// TIA Portal V18 export
FUNCTION_BLOCK "RollerV3"   // FB2, LAD
TITLE = Description:
{ S7_Optimized_Access := 'TRUE' }
VERSION : 0.1
// How to operate and control the roller:
// Roller is controled by inputs in WebDB: Mode, SetSpeed, Direction, OffsetSpeed. To start the roller use Start_Roller and to stop use Stop_Roller.
// 
// Mode descriptions:
// 0 - Controlling the roller by just turning it ON/OFF
// 1 - Basic speed control of the roller with 0-100%
// 2 - Direct speed control based on Y axis velocity. Not useful for printing, but might help in the development process to observe roller system inertia.
// 3 - Setting relative surface velocity (powder to roller). There is no control loop. Could be used for testing the feature before evaluating.
// 
// E-STOP - always check!
// stored: AutoNumber true, IsIECCheckEnabled false, IsRetainMemResEnabled false, MemoryReserve 100, SetENOAutomatically false, UDAEnableTagReadback false
   VAR_INPUT
      "E-STOP" : Bool;
      SystemON : Bool;
      Mode : Int;   // 0 - ON/OFF; 1 - Set Max Speed; 2 - Automatic Yvel=Rvel; 3 - Automatic vel dif
      SetSpeed : Real;   // %
      DirectionLeftRight : Bool;
      Offsetspeed : DInt;
      YAxisVelocity : DInt;
      Roller_HW_address : HW_HSC;
      DoorSensors : Bool;
   END_VAR
   VAR_OUTPUT
      WebDBRollerOutput : Bool;
      RollerDirection : Bool;   // 1 - Clockwise; 0 - Counterclockwise
      RollerLinearVelocity : DInt;   // Microns Per Sec
      RollerRPM : Real;
      RollerRPM_Measured : Real;
   END_VAR
   VAR_IN_OUT
      WebDBStart : Bool;
      WebDBStop : Bool;
   END_VAR
   VAR
      RollerSetReset : Bool;
      RollerFullPower : Bool;
      RollerHalfPower : Bool;
      RollerActive : Bool;
      RollerSpeedInputGeneral { ExternalAccessible := 'False'; ExternalVisible := 'False'; ExternalWritable := 'False'} : Real;   // %
      RollerSpeedInputPID : Real;
      RollerManualValue : Int;
      Direction_Plus { ExternalAccessible := 'False'; ExternalVisible := 'False'; ExternalWritable := 'False'} : Bool;   // Clockwise
      Direction_Minus { ExternalAccessible := 'False'; ExternalVisible := 'False'; ExternalWritable := 'False'} : Bool;   // Counterclockwise
      PulseSignalMeasurement : DWord;
      MaintenanceM3DirDis : Bool := true;
      MaintenanceSkipPID : Bool := true;
      MaintenanceAutomaticDifVel : Bool;   // Change automatic mode from Yvel=Rvel to Difference
      MaintenanceRollerON : Bool;
      RollerDirectionInt_last : Int;
      Roller_RPM_Send_last : Real;
      RollerSetReset_M : Bool;
      RollerSetReset_M2 : Bool;
      hscData : HSC_Period;
   END_VAR
   VAR_TEMP
      DirectionMinusInternal : Bool;
      OffsetSpeedInternal : DInt;
      YAxisVelocityInternal : DInt;
      Roller_Speed_ConvRPM : Real;
      Roller_Speed_ConvPercInput : Real;
      Roller_Speed_ConvDEGSEC : Real;
      Roller_PWM_NormOutput : Real;
      Roller_ConvLinearPerDeg : DInt;
      Roller_Conv_M1_Norm : Real;
      Roller_Conv_M1_Scale : Real;
      Roller_Conv_M2_YvelocityconvRPS : Real;
      Roller_Conv_M2_YvelocityconvRPM : Real;
      Roller_Conv_M3_LinVel : DInt;
      Roller_Conv_M3_Rps : Real;
      Roller_Conv_M3_Rpm : Real;
      Roller_Send_Conv : Real;
      Roller_RPM_Send : Real;
      Roller_RPM_SendRev : Real;
      Roller_Circumference : DInt;   // [microns]
      Roller_Direction_Internal : Bool;
      RollerMinRPMRev : Real;
      RollerDirectionInt : Int;
      ex_vel : Bool;
      RollerDEGPS_send : Real;
      RPMchanged : Bool;
      DirectionChanged : Bool;
      haltAxis : Bool;
   END_VAR
   VAR CONSTANT
      RollerMotorMaxSpeed : Real := 200.0;   // RPM
      MotorToRollerGearRatio : Real := 1.0;   // Belt transmission ratio
      RPMtoDEGSEC : Real := 6.0;   // RPM to Degress per Second conversion factor
      RollerDiameter : DInt := 50000;   // Diameter in microns
      LinearRollerSpeedFactor : Real;   // To convert rotation to linear speed
      RollerPWMPeriod : Int := 10000;
      RollerMinRPM : Real := 5.0;
   END_VAR
   // hscData.EnHSC := TRUE;
   // hscData.EnPeriod := false;
   // hscData.NewPeriod := 1000;
   VAR_TEMP   // added for the SCL form of the ladder/FBD networks
      _w1 : Bool;
      _w2 : Bool;
   END_VAR
BEGIN

REGION Network 1: Roller ON and Speed Control
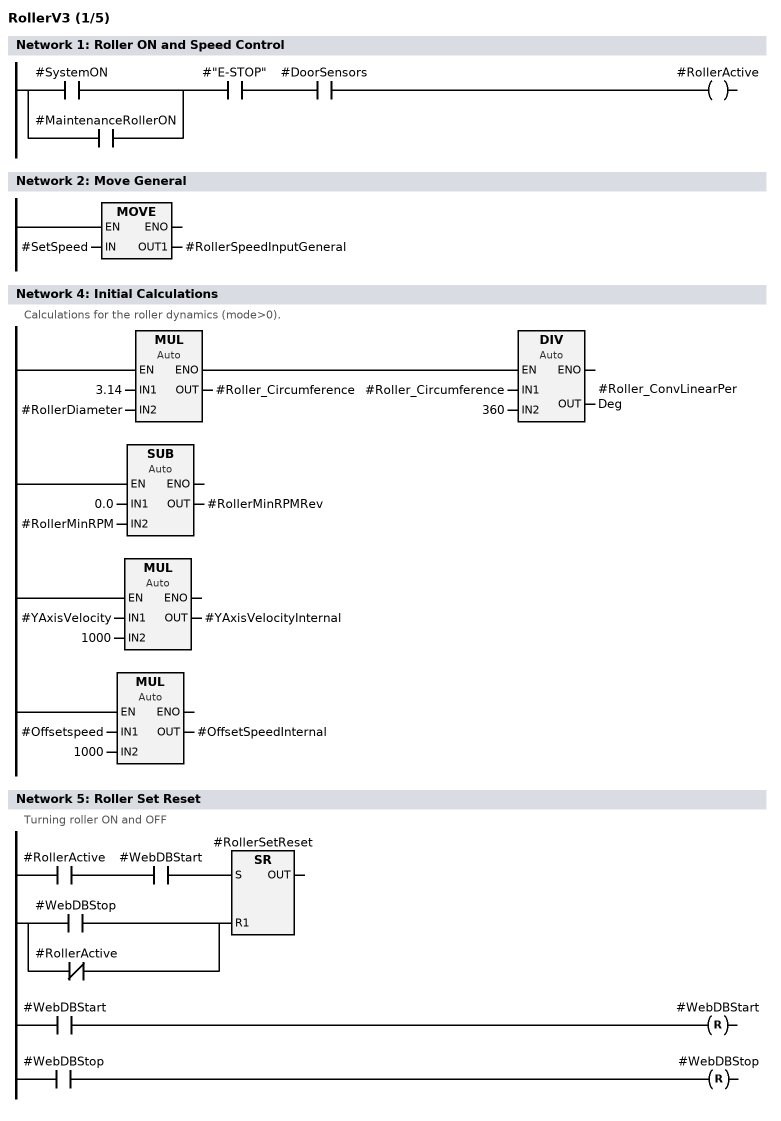
   RUNG wire#powerrail
      Contact( #SystemON )
      wire#w1
      Contact( #"E-STOP" )
      Contact( #DoorSensors )
      Coil( #RollerActive )
   END_RUNG
   RUNG wire#powerrail
      Contact( #MaintenanceRollerON )
   END_RUNG wire#w1
   // the same network as SCL:
   #RollerActive := (#SystemON OR #MaintenanceRollerON) AND #"E-STOP" AND #DoorSensors;
END_REGION

REGION Network 2: Move General
   RUNG wire#powerrail
      Move(in := #SetSpeed, out1 => #RollerSpeedInputGeneral)
   END_RUNG
   // the same network as SCL:
   #RollerSpeedInputGeneral := #SetSpeed;
END_REGION

REGION Network 3: Roller Direction
END_REGION

REGION Network 4: Initial Calculations
   // Calculations for the roller dynamics (mode>0).
   RUNG wire#powerrail
      Mul(in1 := 3.14, in2 := #RollerDiameter, out => #Roller_Circumference)
      Div(in1 := #Roller_Circumference, in2 := 360, out => #Roller_ConvLinearPerDeg)
   END_RUNG
   RUNG wire#powerrail
      Sub(in1 := 0.0, in2 := #RollerMinRPM, out => #RollerMinRPMRev)
   END_RUNG
   RUNG wire#powerrail
      Mul(in1 := #YAxisVelocity, in2 := 1000, out => #YAxisVelocityInternal)
   END_RUNG
   RUNG wire#powerrail
      Mul(in1 := #Offsetspeed, in2 := 1000, out => #OffsetSpeedInternal)
   END_RUNG
   // the same network as SCL:
   #Roller_Circumference := 3.14 * #RollerDiameter;
   #Roller_ConvLinearPerDeg := #Roller_Circumference / 360;
   #RollerMinRPMRev := 0.0 - #RollerMinRPM;
   #YAxisVelocityInternal := #YAxisVelocity * 1000;
   #OffsetSpeedInternal := #Offsetspeed * 1000;
END_REGION

REGION Network 5: Roller Set Reset
   // Turning roller ON and OFF
   RUNG wire#powerrail
      Contact( #RollerActive )
      Contact( #WebDBStart )
      S_SR(operand := #RollerSetReset, r1 := wire#w1)
   END_RUNG
   RUNG wire#powerrail
      Contact( #WebDBStop )
   END_RUNG wire#w1
   RUNG wire#powerrail
      I_Contact( #RollerActive )
   END_RUNG wire#w1
   RUNG wire#powerrail
      Contact( #WebDBStart )
      R_Coil( #WebDBStart )
   END_RUNG
   RUNG wire#powerrail
      Contact( #WebDBStop )
      R_Coil( #WebDBStop )
   END_RUNG
   // the same network as SCL:
   IF #RollerActive AND #WebDBStart THEN
       #RollerSetReset := TRUE;   // SR flip-flop
   END_IF;
   IF #WebDBStop OR NOT #RollerActive THEN #RollerSetReset := FALSE; END_IF;
   IF #WebDBStart THEN #WebDBStart := FALSE; END_IF;
   IF #WebDBStop THEN #WebDBStop := FALSE; END_IF;
END_REGION

REGION Network 6: PID
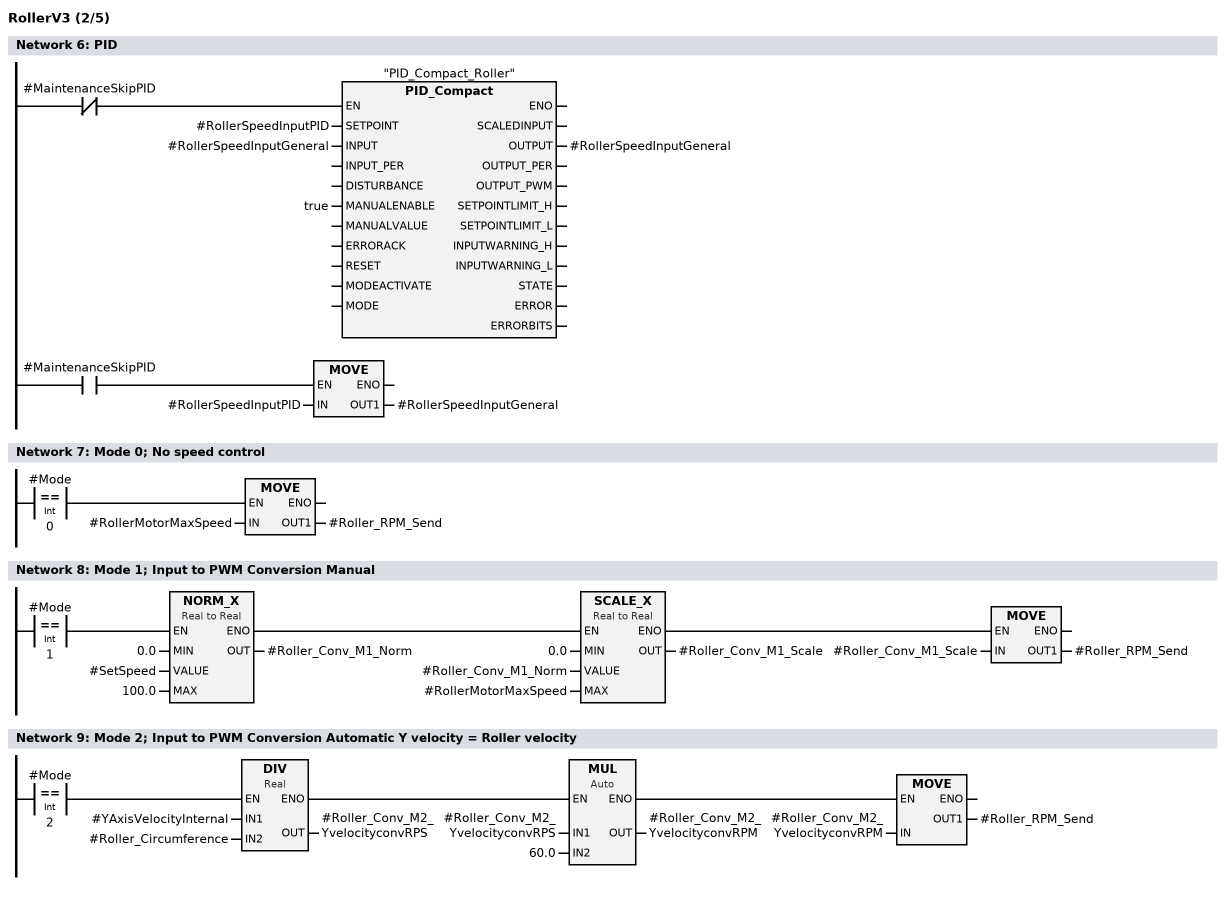
   RUNG wire#powerrail
      I_Contact( #MaintenanceSkipPID )
      "PID_Compact_Roller".PID_Compact(Setpoint := #RollerSpeedInputPID, Input := #RollerSpeedInputGeneral, Input_PER :=, Disturbance :=, ManualEnable := true, ManualValue :=, ErrorAck :=, Reset :=, ModeActivate :=, Mode :=, ScaledInput =>, Output => #RollerSpeedInputGeneral, Output_PER =>, Output_PWM =>, SetpointLimit_H =>, SetpointLimit_L =>, InputWarning_H =>, InputWarning_L =>, State =>, Error =>, ErrorBits =>)
   END_RUNG
   RUNG wire#powerrail
      Contact( #MaintenanceSkipPID )
      Move(in := #RollerSpeedInputPID, out1 => #RollerSpeedInputGeneral)
   END_RUNG
   // the same network as SCL:
   IF NOT #MaintenanceSkipPID THEN
       "PID_Compact_Roller"(Setpoint := #RollerSpeedInputPID,   // PID_Compact
                            Input := #RollerSpeedInputGeneral,
                            ManualEnable := true,
                            Output => #RollerSpeedInputGeneral);
   END_IF;
   IF #MaintenanceSkipPID THEN #RollerSpeedInputGeneral := #RollerSpeedInputPID; END_IF;
END_REGION

REGION Network 7: Mode 0; No speed control
   RUNG wire#powerrail
      { S7_Templates := "SrcType := Int" } EQ_Contact(in1 := #Mode, in2 := 0)
      Move(in := #RollerMotorMaxSpeed, out1 => #Roller_RPM_Send)
   END_RUNG
   // the same network as SCL:
   IF #Mode = 0 THEN #Roller_RPM_Send := #RollerMotorMaxSpeed; END_IF;
END_REGION

REGION Network 8: Mode 1; Input to PWM Conversion Manual
   RUNG wire#powerrail
      { S7_Templates := "SrcType := Int" } EQ_Contact(in1 := #Mode, in2 := 1)
      { S7_Templates := "[SrcType := Real, DestType := Real]" } Normalize(min := 0.0, value := #SetSpeed, max := 100.0, out => #Roller_Conv_M1_Norm)
      { S7_Templates := "[SrcType := Real, DestType := Real]" } Scale(min := 0.0, value := #Roller_Conv_M1_Norm, max := #RollerMotorMaxSpeed, out => #Roller_Conv_M1_Scale)
      Move(in := #Roller_Conv_M1_Scale, out1 => #Roller_RPM_Send)
   END_RUNG
   // the same network as SCL:
   IF #Mode = 1 THEN
       #Roller_Conv_M1_Norm := NORM_X(MIN := 0.0, VALUE := #SetSpeed, MAX := 100.0);
       #Roller_Conv_M1_Scale := SCALE_X(MIN := 0.0, VALUE := #Roller_Conv_M1_Norm, MAX := #RollerMotorMaxSpeed);
       #Roller_RPM_Send := #Roller_Conv_M1_Scale;
   END_IF;
END_REGION

REGION Network 9: Mode 2; Input to PWM Conversion Automatic Y velocity = Roller velocity
   RUNG wire#powerrail
      { S7_Templates := "SrcType := Int" } EQ_Contact(in1 := #Mode, in2 := 2)
      { S7_Templates := "SrcType := Real" } Div(in1 := #YAxisVelocityInternal, in2 := #Roller_Circumference, out => #Roller_Conv_M2_YvelocityconvRPS)
      Mul(in1 := #Roller_Conv_M2_YvelocityconvRPS, in2 := 60.0, out => #Roller_Conv_M2_YvelocityconvRPM)
      Move(in := #Roller_Conv_M2_YvelocityconvRPM, out1 => #Roller_RPM_Send)
   END_RUNG
   // the same network as SCL:
   IF #Mode = 2 THEN
       #Roller_Conv_M2_YvelocityconvRPS := #YAxisVelocityInternal / #Roller_Circumference;
       #Roller_Conv_M2_YvelocityconvRPM := #Roller_Conv_M2_YvelocityconvRPS * 60.0;
       #Roller_RPM_Send := #Roller_Conv_M2_YvelocityconvRPM;
   END_IF;
END_REGION

REGION Network 10: Mode 3; Input to PWM Conversion Setting Speed Difference according to the Y velocity
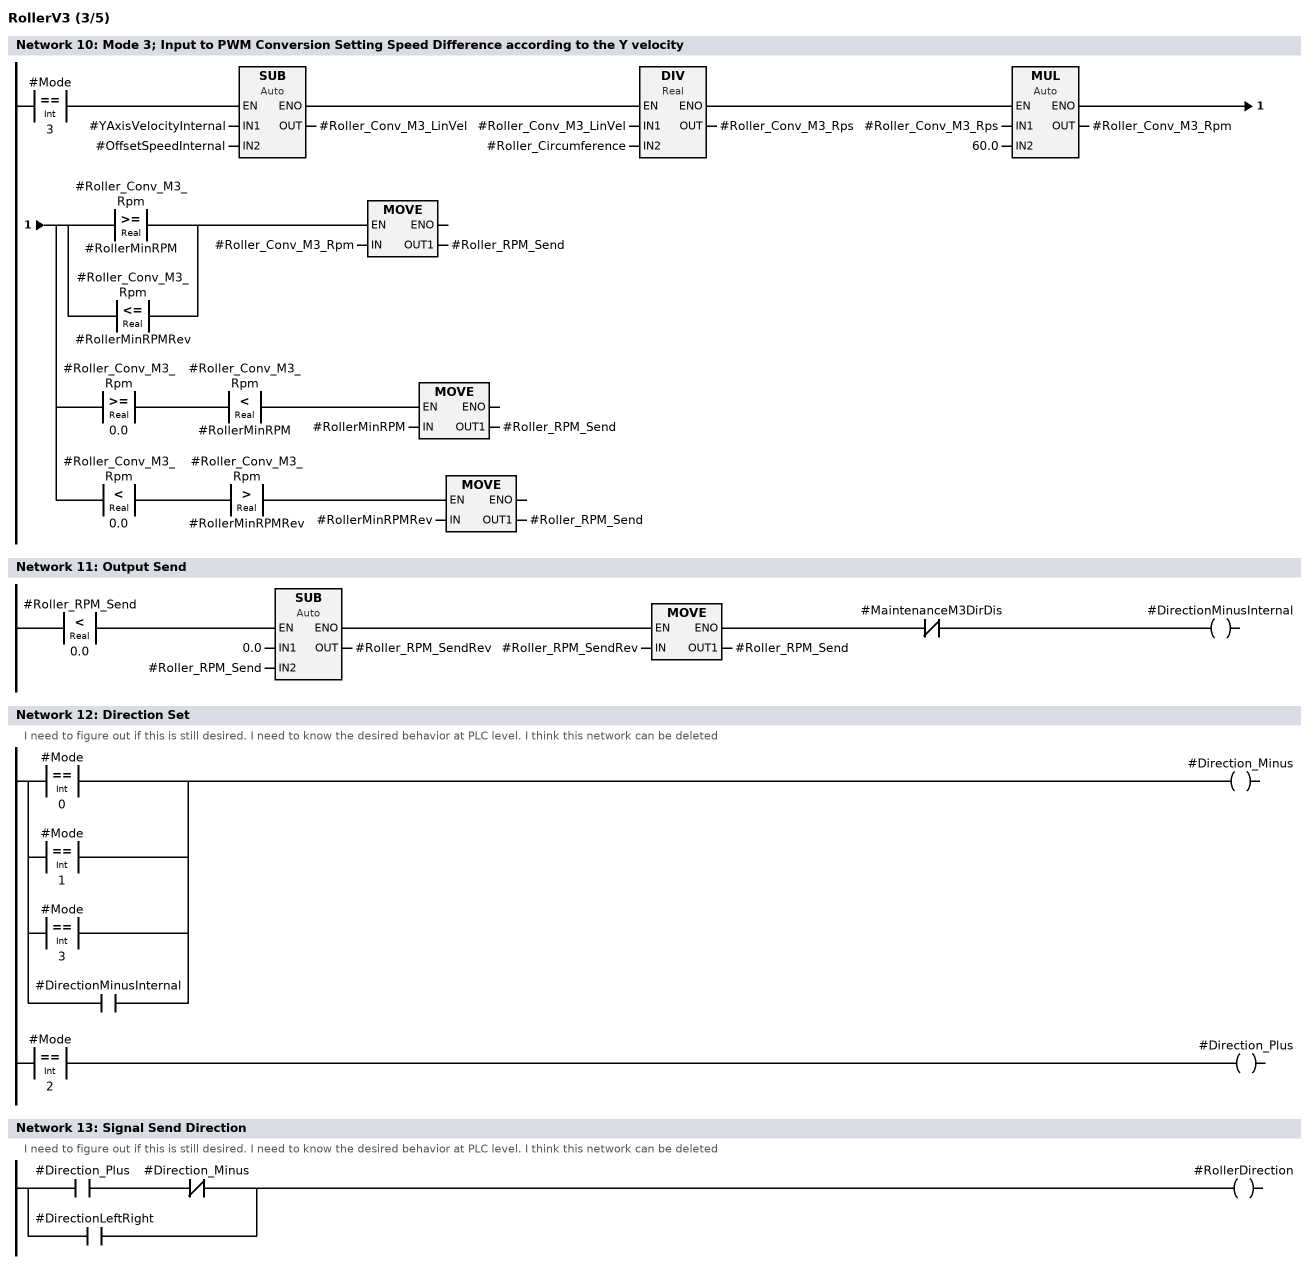
   RUNG wire#powerrail
      { S7_Templates := "SrcType := Int" } EQ_Contact(in1 := #Mode, in2 := 3)
      Sub(in1 := #YAxisVelocityInternal, in2 := #OffsetSpeedInternal, out => #Roller_Conv_M3_LinVel)
      { S7_Templates := "SrcType := Real" } Div(in1 := #Roller_Conv_M3_LinVel, in2 := #Roller_Circumference, out => #Roller_Conv_M3_Rps)
      Mul(in1 := #Roller_Conv_M3_Rps, in2 := 60.0, out => #Roller_Conv_M3_Rpm)
      wire#w1
      { S7_Templates := "SrcType := Real" } GE_Contact(in1 := #Roller_Conv_M3_Rpm, in2 := #RollerMinRPM)
      wire#w2
      Move(in := #Roller_Conv_M3_Rpm, out1 => #Roller_RPM_Send)
   END_RUNG
   RUNG wire#w1
      { S7_Templates := "SrcType := Real" } LE_Contact(in1 := #Roller_Conv_M3_Rpm, in2 := #RollerMinRPMRev)
   END_RUNG wire#w2
   RUNG wire#w1
      { S7_Templates := "SrcType := Real" } GE_Contact(in1 := #Roller_Conv_M3_Rpm, in2 := 0.0)
      { S7_Templates := "SrcType := Real" } LT_Contact(in1 := #Roller_Conv_M3_Rpm, in2 := #RollerMinRPM)
      Move(in := #RollerMinRPM, out1 => #Roller_RPM_Send)
   END_RUNG
   RUNG wire#w1
      { S7_Templates := "SrcType := Real" } LT_Contact(in1 := #Roller_Conv_M3_Rpm, in2 := 0.0)
      { S7_Templates := "SrcType := Real" } GT_Contact(in1 := #Roller_Conv_M3_Rpm, in2 := #RollerMinRPMRev)
      Move(in := #RollerMinRPMRev, out1 => #Roller_RPM_Send)
   END_RUNG
   // the same network as SCL:
   #_w1 := #Mode = 3;
   IF #_w1 THEN
       #Roller_Conv_M3_LinVel := #YAxisVelocityInternal - #OffsetSpeedInternal;
       #Roller_Conv_M3_Rps := #Roller_Conv_M3_LinVel / #Roller_Circumference;
       #Roller_Conv_M3_Rpm := #Roller_Conv_M3_Rps * 60.0;
   END_IF;
   IF #_w1 AND ((#Roller_Conv_M3_Rpm >= #RollerMinRPM) OR (#Roller_Conv_M3_Rpm <= #RollerMinRPMRev)) THEN
       #Roller_RPM_Send := #Roller_Conv_M3_Rpm;
   END_IF;
   IF #_w1 AND (#Roller_Conv_M3_Rpm >= 0.0) AND (#Roller_Conv_M3_Rpm < #RollerMinRPM) THEN
       #Roller_RPM_Send := #RollerMinRPM;
   END_IF;
   IF #_w1 AND (#Roller_Conv_M3_Rpm < 0.0) AND (#Roller_Conv_M3_Rpm > #RollerMinRPMRev) THEN
       #Roller_RPM_Send := #RollerMinRPMRev;
   END_IF;
END_REGION

REGION Network 11: Output Send
   RUNG wire#powerrail
      { S7_Templates := "SrcType := Real" } LT_Contact(in1 := #Roller_RPM_Send, in2 := 0.0)
      Sub(in1 := 0.0, in2 := #Roller_RPM_Send, out => #Roller_RPM_SendRev)
      Move(in := #Roller_RPM_SendRev, out1 => #Roller_RPM_Send)
      I_Contact( #MaintenanceM3DirDis )
      Coil( #DirectionMinusInternal )
   END_RUNG
   // the same network as SCL:
   #_w1 := #Roller_RPM_Send < 0.0;
   IF #_w1 THEN
       #Roller_RPM_SendRev := 0.0 - #Roller_RPM_Send;
       #Roller_RPM_Send := #Roller_RPM_SendRev;
   END_IF;
   #DirectionMinusInternal := #_w1 AND NOT #MaintenanceM3DirDis;
END_REGION

REGION Network 12: Direction Set
   // I need to figure out if this is still desired. I need to know the desired behavior at PLC level. I think this network can be deleted
   RUNG wire#powerrail
      { S7_Templates := "SrcType := Int" } EQ_Contact(in1 := #Mode, in2 := 0)
      wire#w1
      Coil( #Direction_Minus )
   END_RUNG
   RUNG wire#powerrail
      { S7_Templates := "SrcType := Int" } EQ_Contact(in1 := #Mode, in2 := 1)
   END_RUNG wire#w1
   RUNG wire#powerrail
      { S7_Templates := "SrcType := Int" } EQ_Contact(in1 := #Mode, in2 := 3)
   END_RUNG wire#w1
   RUNG wire#powerrail
      Contact( #DirectionMinusInternal )
   END_RUNG wire#w1
   RUNG wire#powerrail
      { S7_Templates := "SrcType := Int" } EQ_Contact(in1 := #Mode, in2 := 2)
      Coil( #Direction_Plus )
   END_RUNG
   // the same network as SCL:
   #Direction_Minus := (#Mode = 0) OR (#Mode = 1) OR (#Mode = 3) OR #DirectionMinusInternal;
   #Direction_Plus := #Mode = 2;
END_REGION

REGION Network 13: Signal Send Direction
   // I need to figure out if this is still desired. I need to know the desired behavior at PLC level. I think this network can be deleted
   RUNG wire#powerrail
      Contact( #Direction_Plus )
      I_Contact( #Direction_Minus )
      wire#w1
      Coil( #RollerDirection )
   END_RUNG
   RUNG wire#powerrail
      Contact( #DirectionLeftRight )
   END_RUNG wire#w1
   // the same network as SCL:
   #RollerDirection := (#Direction_Plus AND NOT #Direction_Minus) OR #DirectionLeftRight;
END_REGION

REGION Network 14
   // Convert Rotations per minute to degrees per second, as the technology object works with degrees. First, copy RPM send to an output variable, for output/logging purposes.
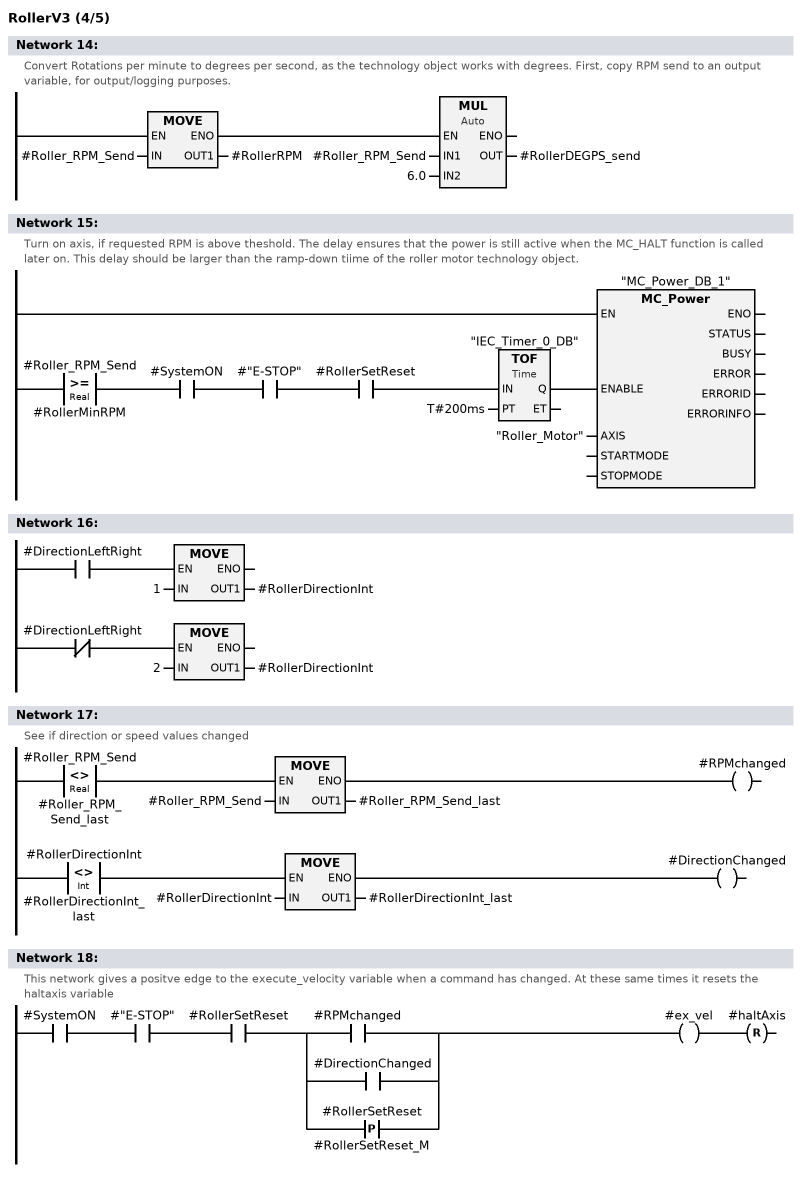
   RUNG wire#powerrail
      Move(in := #Roller_RPM_Send, out1 => #RollerRPM)
      Mul(in1 := #Roller_RPM_Send, in2 := 6.0, out => #RollerDEGPS_send)
   END_RUNG
   // the same network as SCL:
   #RollerRPM := #Roller_RPM_Send;
   #RollerDEGPS_send := #Roller_RPM_Send * 6.0;
END_REGION

REGION Network 15
   // Turn on axis, if requested RPM is above theshold. The delay ensures that the power is still active when the MC_HALT function is called later on. This delay should be larger than the ramp-down tiime of the roller motor technology object.
   RUNG wire#powerrail
      "MC_Power_DB_1".MC_Power(Enable := wire#w1, Axis := "Roller_Motor", StartMode :=, StopMode :=, Status =>, Busy =>, Error =>, ErrorID =>, ErrorInfo =>)
   END_RUNG
   RUNG wire#powerrail
      { S7_Templates := "SrcType := Real" } GE_Contact(in1 := #Roller_RPM_Send, in2 := #RollerMinRPM)
      Contact( #SystemON )
      Contact( #"E-STOP" )
      Contact( #RollerSetReset )
      { S7_Templates := "time_type := Time" } "IEC_Timer_0_DB".TOF(pt := T#200ms, et =>)
   END_RUNG wire#w1
   // the same network as SCL:
   "IEC_Timer_0_DB".TOF(IN := (#Roller_RPM_Send >= #RollerMinRPM) AND #SystemON AND #"E-STOP" AND #RollerSetReset,
                        PT := T#200ms);
   "MC_Power_DB_1"(Enable := "IEC_Timer_0_DB".Q, Axis := "Roller_Motor");   // MC_Power
END_REGION

REGION Network 16
   RUNG wire#powerrail
      Contact( #DirectionLeftRight )
      Move(in := 1, out1 => #RollerDirectionInt)
   END_RUNG
   RUNG wire#powerrail
      I_Contact( #DirectionLeftRight )
      Move(in := 2, out1 => #RollerDirectionInt)
   END_RUNG
   // the same network as SCL:
   IF #DirectionLeftRight THEN #RollerDirectionInt := 1; END_IF;
   IF NOT #DirectionLeftRight THEN #RollerDirectionInt := 2; END_IF;
END_REGION

REGION Network 17
   // See if direction or speed values changed
   RUNG wire#powerrail
      { S7_Templates := "SrcType := Real" } NE_Contact(in1 := #Roller_RPM_Send, in2 := #Roller_RPM_Send_last)
      Move(in := #Roller_RPM_Send, out1 => #Roller_RPM_Send_last)
      Coil( #RPMchanged )
   END_RUNG
   RUNG wire#powerrail
      { S7_Templates := "SrcType := Int" } NE_Contact(in1 := #RollerDirectionInt, in2 := #RollerDirectionInt_last)
      Move(in := #RollerDirectionInt, out1 => #RollerDirectionInt_last)
      Coil( #DirectionChanged )
   END_RUNG
   // the same network as SCL:
   #_w1 := #Roller_RPM_Send <> #Roller_RPM_Send_last;
   IF #_w1 THEN #Roller_RPM_Send_last := #Roller_RPM_Send; END_IF;
   #RPMchanged := #_w1;
   #_w2 := #RollerDirectionInt <> #RollerDirectionInt_last;
   IF #_w2 THEN #RollerDirectionInt_last := #RollerDirectionInt; END_IF;
   #DirectionChanged := #_w2;
END_REGION

REGION Network 18
   // This network gives a positve edge to the execute_velocity variable when a command has changed. At these same times it resets the haltaxis variable
   RUNG wire#powerrail
      Contact( #SystemON )
      Contact( #"E-STOP" )
      Contact( #RollerSetReset )
      wire#w1
      Contact( #RPMchanged )
      wire#w2
      Coil( #ex_vel )
      R_Coil( #haltAxis )
   END_RUNG
   RUNG wire#w1
      Contact( #DirectionChanged )
   END_RUNG wire#w2
   RUNG wire#w1
      P_Contact(operand := #RollerSetReset, bit := #RollerSetReset_M)
   END_RUNG wire#w2
   // the same network as SCL:
   #_w1 := #SystemON AND #"E-STOP" AND #RollerSetReset AND #RollerSetReset AND NOT #RollerSetReset_M;   // rising edge of #RollerSetReset
   #RollerSetReset_M := #RollerSetReset;
   #ex_vel := (#SystemON AND #"E-STOP" AND #RollerSetReset AND (#RPMchanged OR #DirectionChanged)) OR #_w1;
   IF #ex_vel THEN #haltAxis := FALSE; END_IF;
END_REGION

REGION Network 19: Convert dircetion command to INT; Send command to drive
   // Direction; 0 means that the direction is in the sigh of the velocity; 1 is positive direction; 2 is negative direction
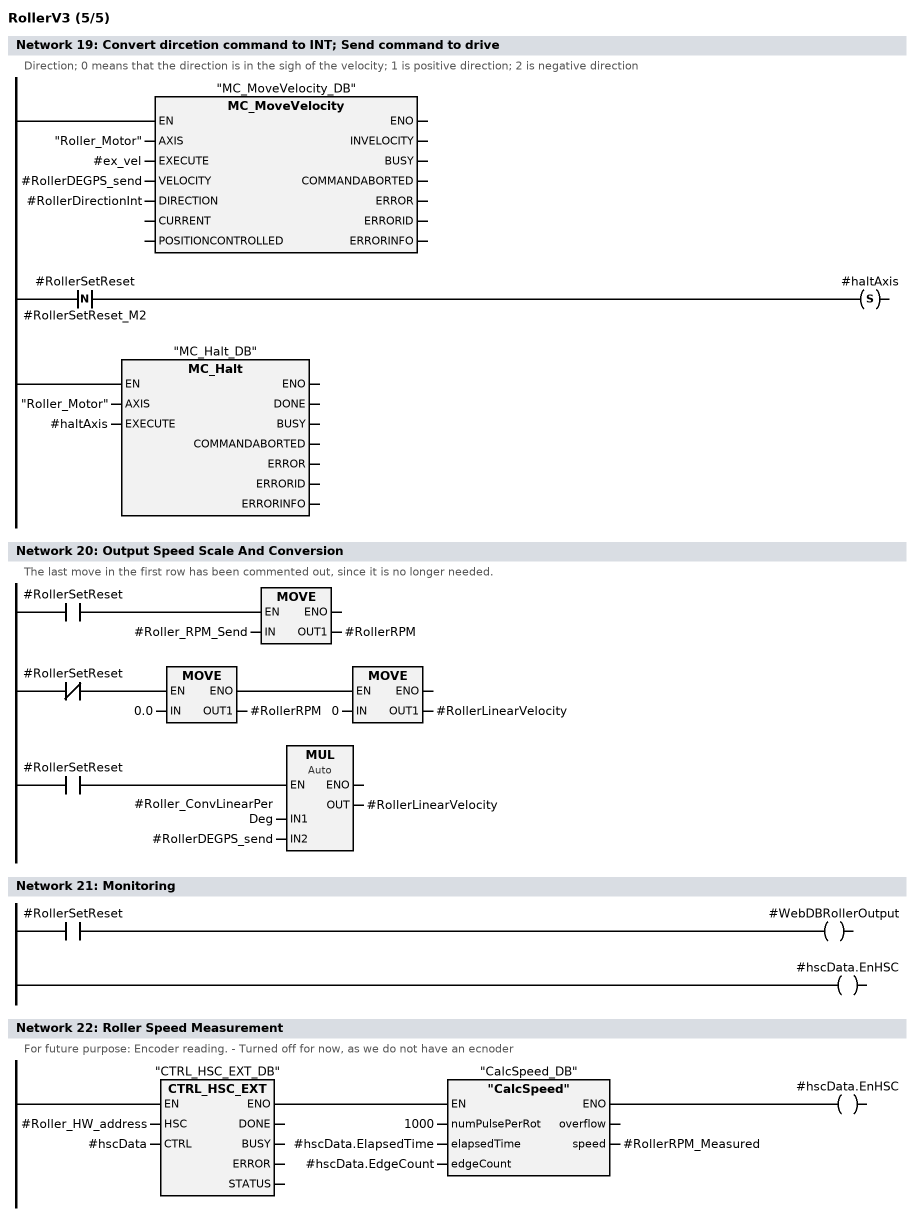
   RUNG wire#powerrail
      "MC_MoveVelocity_DB".MC_MoveVelocity(Axis := "Roller_Motor", Execute := #ex_vel, Velocity := #RollerDEGPS_send, Direction := #RollerDirectionInt, Current :=, PositionControlled :=, InVelocity =>, Busy =>, CommandAborted =>, Error =>, ErrorID =>, ErrorInfo =>)
   END_RUNG
   RUNG wire#powerrail
      N_Contact(operand := #RollerSetReset, bit := #RollerSetReset_M2)
      S_Coil( #haltAxis )
   END_RUNG
   RUNG wire#powerrail
      "MC_Halt_DB".MC_Halt(Axis := "Roller_Motor", Execute := #haltAxis, Done =>, Busy =>, CommandAborted =>, Error =>, ErrorID =>, ErrorInfo =>)
   END_RUNG
   // the same network as SCL:
   "MC_MoveVelocity_DB"(Axis := "Roller_Motor",   // MC_MoveVelocity
                        Execute := #ex_vel,
                        Velocity := #RollerDEGPS_send,
                        Direction := #RollerDirectionInt);
   #_w1 := NOT #RollerSetReset AND #RollerSetReset_M2;   // falling edge of #RollerSetReset
   #RollerSetReset_M2 := #RollerSetReset;
   IF #_w1 THEN #haltAxis := TRUE; END_IF;
   "MC_Halt_DB"(Axis := "Roller_Motor", Execute := #haltAxis);   // MC_Halt
END_REGION

REGION Network 20: Output Speed Scale And Conversion
   // The last move in the first row has been commented out, since it is no longer needed.
   RUNG wire#powerrail
      Contact( #RollerSetReset )
      Move(in := #Roller_RPM_Send, out1 => #RollerRPM)
   END_RUNG
   RUNG wire#powerrail
      I_Contact( #RollerSetReset )
      Move(in := 0.0, out1 => #RollerRPM)
      Move(in := 0, out1 => #RollerLinearVelocity)
   END_RUNG
   RUNG wire#powerrail
      Contact( #RollerSetReset )
      Mul(in1 := #Roller_ConvLinearPerDeg, in2 := #RollerDEGPS_send, out => #RollerLinearVelocity)
   END_RUNG
   // the same network as SCL:
   IF #RollerSetReset THEN #RollerRPM := #Roller_RPM_Send; END_IF;
   IF NOT #RollerSetReset THEN
       #RollerRPM := 0.0;
       #RollerLinearVelocity := 0;
   END_IF;
   IF #RollerSetReset THEN #RollerLinearVelocity := #Roller_ConvLinearPerDeg * #RollerDEGPS_send; END_IF;
END_REGION

REGION Network 21: Monitoring
   RUNG wire#powerrail
      Contact( #RollerSetReset )
      Coil( #WebDBRollerOutput )
   END_RUNG
   RUNG wire#powerrail
      Coil( #hscData.EnHSC )
   END_RUNG
   // the same network as SCL:
   #WebDBRollerOutput := #RollerSetReset;
   #hscData.EnHSC := TRUE;
END_REGION

REGION Network 22: Roller Speed Measurement
   // For future purpose: Encoder reading. - Turned off for now, as we do not have an ecnoder
   RUNG wire#powerrail
      "CTRL_HSC_EXT_DB".CTRL_HSC_EXT(HSC := #Roller_HW_address, CTRL := #hscData, DONE =>, BUSY =>, ERROR =>, STATUS =>)
      "CalcSpeed_DB"(numPulsePerRot := 1000, elapsedTime := #hscData.ElapsedTime, edgeCount := #hscData.EdgeCount, overflow =>, speed => #RollerRPM_Measured)
      Coil( #hscData.EnHSC )
   END_RUNG
   // the same network as SCL:
   "CTRL_HSC_EXT_DB"(HSC := #Roller_HW_address, CTRL := #hscData, ENO => #_w1);   // CTRL_HSC_EXT
   "CalcSpeed_DB"(EN := #_w1,   // "CalcSpeed"
                  numPulsePerRot := 1000,
                  elapsedTime := #hscData.ElapsedTime,
                  edgeCount := #hscData.EdgeCount,
                  speed => #RollerRPM_Measured,
                  ENO => #_w2);
   #hscData.EnHSC := #_w2;
END_REGION
END_FUNCTION_BLOCK
